// TIA Portal V16 export
// export: Created 2021-04-16T08:36:19.4507438Z, ExportSetting WithDefaults, DisplayName Totally Integrated Automation Portal, DisplayVersion V16 Update 3, DisplayName TIA Portal Version Control Interface, DisplayVersion V16 Update 2, DisplayName TIA Portal Openness, DisplayVersion V16 Update 3, DisplayName SINAMICS Startdrive Advanced, DisplayVersion V16 Update 5, DisplayName SINAMICS Startdrive G130, G150, S120, S150, SINAMICS MV, S210, DisplayVersion V16 Update 5, DisplayName SINAMICS Startdrive G110M, G120, G120C, G120D, G120P, G115D, DisplayVersion V16 Update 5, DisplayName STEP 7 Professional, DisplayVersion V16 Update 3, DisplayName STEP 7 Safety, DisplayVersion V16, DisplayName WinCC Professional, DisplayVersion V16 Update 3
FUNCTION "Test_AWL" : Void   // FC2, STL
{ S7_Optimized_Access := 'TRUE' }
VERSION : 0.1
// stored: AutoNumber true, UDAEnableTagReadback false
   VAR_TEMP
      x_Test_1 : Bool;
      x_Test_2 : Bool;
      x_Test_3 : Bool;
      x_Test_4 : Bool;
      x_Test_5 : Bool;
   END_VAR
BEGIN

NETWORK
TITLE = 
      A     #x_Test_1;
      =     #x_Test_2;

END_FUNCTION
